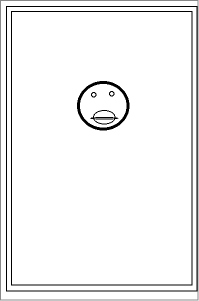
VISUALIZATION Elevator  // 199x301
    Rectangle (6,6 191x285)
    Rectangle (11,11 181x274)
    Ellipse (77,81 52x49)
    Polyline (117,230)
    Polyline (151,299)
    Polyline (81,297)
    Polyline (165,151)
    Polyline (73,152)
    Ellipse (93,110 22x14), invisible if: NOT Process.xMotorRunning
    Ellipse (91,92 5x5)
    Ellipse (109,91 5x5)
    Ellipse (90,117 28x2), invisible if: Process.xMotorRunning
END_VISUALIZATION

(* stored: Version 1.1.0.1, ProductVersion 3.1.4024.12
   Visu Elevator: Id {23d5df2b-296e-4146-9958-04cbe38054df} *)
